// TwinCAT 3 PLC project Main
// ProgramVersion: 3.1.4022.4
// libraries:
//   Tc2_FTP, * (Beckhoff Automation GmbH)
//   Tc2_MC2, * (Beckhoff Automation GmbH)
//   Tc2_NCI, * (Beckhoff Automation GmbH)
//   Tc2_Standard, * (Beckhoff Automation GmbH)
//   Tc2_System, * (Beckhoff Automation GmbH)
//   Tc2_Utilities, * (Beckhoff Automation GmbH)
//   Tc3_IotBase, * (Beckhoff Automation GmbH)
//   Tc3_JsonXml, * (Beckhoff Automation GmbH)
//   Tc3_Module, * (Beckhoff Automation GmbH)
//   VisuSymbols,3.5.10.0,System
// project tree:
//   / GlobalTextList.TcGTLO, PlcTask.TcTTO, Visualization Manager.TcVMO (not stored)
//   GVLs/ COM.TcGVL, gcode.TcGVL, GVL.TcGVL
//   POUs/COMMANDS/ commandDecoder.TcPOU, commandExecute.TcPOU, POU_NCI.TcPOU
//   POUs/ ERROR.TcPOU, knoppen.TcPOU, MAIN_XYZ.TcPOU
//   POUs/JSON/ decCOM.TcPOU, decCOM_PLC.TcPOU, decFile.TcPOU, readJSONfile.TcPOU
//   POUs/MQTT/ MAIN_MQTT.TcPOU, PrgMqttCom.TcPOU, SubMqttCom.TcPOU
//   VISUs/ Basic.TcVIS, bStopAll.TcVIS, vKnoppen.TcVIS
// real-time tasks:
//   TASK PlcTask: cycle T#10ms, priority 20, ADS port 350
// motion (NC):
//   TASK NC-Task 1 SAF: cycle T#2ms, priority 4, ADS port 501
//   TASK NC-Task 1 SVB: cycle T#10ms, priority 8, ADS port 511
//   AXIS Axis X1 (id 1)
//     OtherSettings: AllowMotionCmdToSlave=true
//     encoder EncType=4
//       EncPara: ScaleFactorNumerator=40, ScaleFactorDenominator=12800, Inverse=true, MaxCount=#x0000ffff
//         SoftEndMinControl: Enable=true
//         SoftEndMaxControl: Enable=true, Range=275
//         Inc: RefSearchInverse=true, RefSyncInverse=false, RefMode=1, RefSoftSyncMask=#x0000ffff
//     drive DrvType=24
//       DrvPara: Inverse=true
//         Analog: VeloReferenz=400, ScaleFactorActTorque=0.1
//         TimeComp: TaskDelayCycles=1
//     controller CtrType=1
//       CtrPara: PriorControlFactor=1
//         PID: PosKp=25
//         Observer: BandWidth=20
//   AXIS Axis X2 (id 2)
//     OtherSettings: AllowMotionCmdToSlave=true
//     encoder EncType=4
//       EncPara: ScaleFactorNumerator=40, ScaleFactorDenominator=12800, Inverse=true, MaxCount=#x0000ffff
//         Inc: RefSoftSyncMask=#x0000ffff
//     drive DrvType=24
//       DrvPara: Inverse=true
//         Analog: VeloReferenz=400, ScaleFactorActTorque=0.1
//         TimeComp: TaskDelayCycles=1
//     controller CtrType=1
//       CtrPara: PriorControlFactor=1
//         PID: PosKp=25
//         Observer: BandWidth=20
//   AXIS Axis Y (id 4)
//     OtherSettings: AllowMotionCmdToSlave=true
//     encoder EncType=4
//       EncPara: ScaleFactorNumerator=40, ScaleFactorDenominator=12800, Inverse=true, MaxCount=#x0000ffff
//         SoftEndMinControl: Enable=true
//         SoftEndMaxControl: Enable=true, Range=275
//         Inc: RefSearchInverse=true, RefSyncInverse=false, RefMode=1, RefSoftSyncMask=#x0000ffff
//     drive DrvType=24
//       DrvPara: Inverse=true
//         Analog: VeloReferenz=400, ScaleFactorActTorque=0.1
//         TimeComp: TaskDelayCycles=1
//     controller CtrType=1
//       CtrPara: PriorControlFactor=1
//         PID: PosKp=25
//         Observer: BandWidth=20
//   AXIS Axis Z (id 3)
//     Velo: SlowManual=2, FastManual=5
//     OtherSettings: AllowMotionCmdToSlave=true
//     encoder EncType=4
//       EncPara: ScaleFactorNumerator=1, ScaleFactorDenominator=12800, MaxCount=#x0000ffff
//         Inc: RefSoftSyncMask=#x0000ffff
//     drive DrvType=24
//       Analog: VeloReferenz=10, ScaleFactorActTorque=0.1
//       TimeComp: TaskDelayCycles=1
//     controller CtrType=1
//       CtrPara: PriorControlFactor=1
//         PID: PosKp=25
//         Observer: BandWidth=20
// I/O:
//   DEVICE Device 3 (EtherCAT), AmsNetId 192.168.0.108.4.1
//     Term 1 (EK1100) [EK1100 EtherCAT Coupler (2A E-Bus)]
//       Term 2 (EL7031-0030) [EL7031-0030 1Ch. Stepper motor output stage (24V, 2.8A)]
//       Term 3 (EL7031-0030) [EL7031-0030 1Ch. Stepper motor output stage (24V, 2.8A)]
//       Term 4 (EL7031-0030) [EL7031-0030 1Ch. Stepper motor output stage (24V, 2.8A)]
//       Term 5 (EL7031-0030) [EL7031-0030 1Ch. Stepper motor output stage (24V, 2.8A)]
//       Term 6 (EL1008) [EL1008 8Ch. Dig. Input 24V, 3ms]
//       Term 14 (EL2008) [EL2008 8Ch. Dig. Output 24V, 0.5A]
//       Term 15 (EL3062) [EL3062 2Ch. Ana. Input 0-10V]
//       Term 7 (EL9011) [EL9011 End Terminal]
// variable links:
//   NC-Task 1 SAF/Axes/Axis X1 <-> Device 3 (EtherCAT)/Term 1 (EK1100)/Term 2 (EL7031-0030)
//     Drive/Inputs/In/nState1 @bit 3 <-> STM Status/Status/Error
//     Drive/Inputs/In/nState1 @bit 5 <-> STM Status/Status/Moving negative
//     Drive/Inputs/In/nState1 @bit 4 <-> STM Status/Status/Moving positive
//     Drive/Inputs/In/nState1 @bit 1 <-> STM Status/Status/Ready
//     Drive/Inputs/In/nState1 <-> STM Status/Status/Ready to enable
//     Drive/Inputs/In/nState1 @bit 6 <-> STM Status/Status/Torque reduced
//     Drive/Inputs/In/nState1 @bit 2 <-> STM Status/Status/Warning
//     Drive/Inputs/In/nState2 @bit 3 <-> STM Status/Status/Digital input 1
//     Drive/Inputs/In/nState2 @bit 4 <-> STM Status/Status/Digital input 2
//     Drive/Inputs/In/nState2 @bit 5 <-> STM Status/Status/Sync error
//     Drive/Inputs/In/nState2 @bit 7 <-> STM Status/Status/TxPDO Toggle
//     Drive/Inputs/In/nState4 @bit 1 <-> WcState/InputToggle
//     Drive/Inputs/In/nState4 <-> WcState/WcState
//     Drive/Outputs/Out/nCtrl1 <-> STM Control/Control/Enable
//     Drive/Outputs/Out/nCtrl1 @bit 2 <-> STM Control/Control/Reduce torque
//     Drive/Outputs/Out/nCtrl1 @bit 1 <-> STM Control/Control/Reset
//     Drive/Outputs/Out/nDataOut2[0] <-> STM Velocity/Velocity
//     Enc/Inputs/In/nDataIn1[0] <-> ENC Status compact/Counter value
//     Enc/Inputs/In/nDataIn2[0] <-> ENC Status compact/Latch value
//     Enc/Inputs/In/nState1 @bit 4 <-> ENC Status compact/Status/Counter overflow
//     Enc/Inputs/In/nState1 @bit 3 <-> ENC Status compact/Status/Counter underflow
//     Enc/Inputs/In/nState1 @bit 1 <-> ENC Status compact/Status/Latch extern valid
//     Enc/Inputs/In/nState1 @bit 2 <-> ENC Status compact/Status/Set counter done
//     Enc/Inputs/In/nState2 @bit 4 <-> ENC Status compact/Status/Status of extern latch
//     Enc/Inputs/In/nState2 @bit 5 <-> ENC Status compact/Status/Sync error
//     Enc/Inputs/In/nState2 @bit 7 <-> ENC Status compact/Status/TxPDO Toggle
//     Enc/Inputs/In/nState4 @bit 1 <-> WcState/InputToggle
//     Enc/Inputs/In/nState4 <-> WcState/WcState
//     Enc/Outputs/Out/nCtrl1 @bit 3 <-> ENC Control compact/Control/Enable latch extern on negative edge
//     Enc/Outputs/Out/nCtrl1 @bit 1 <-> ENC Control compact/Control/Enable latch extern on positive edge
//     Enc/Outputs/Out/nCtrl1 @bit 2 <-> ENC Control compact/Control/Set counter
//     Enc/Outputs/Out/nDataOut1[0] <-> ENC Control compact/Set counter value
//   NC-Task 1 SAF/Axes/Axis X2 <-> Device 3 (EtherCAT)/Term 1 (EK1100)/Term 3 (EL7031-0030)
//     Drive/Inputs/In/nState1 @bit 3 <-> STM Status/Status/Error
//     Drive/Inputs/In/nState1 @bit 5 <-> STM Status/Status/Moving negative
//     Drive/Inputs/In/nState1 @bit 4 <-> STM Status/Status/Moving positive
//     Drive/Inputs/In/nState1 @bit 1 <-> STM Status/Status/Ready
//     Drive/Inputs/In/nState1 <-> STM Status/Status/Ready to enable
//     Drive/Inputs/In/nState1 @bit 6 <-> STM Status/Status/Torque reduced
//     Drive/Inputs/In/nState1 @bit 2 <-> STM Status/Status/Warning
//     Drive/Inputs/In/nState2 @bit 3 <-> STM Status/Status/Digital input 1
//     Drive/Inputs/In/nState2 @bit 4 <-> STM Status/Status/Digital input 2
//     Drive/Inputs/In/nState2 @bit 5 <-> STM Status/Status/Sync error
//     Drive/Inputs/In/nState2 @bit 7 <-> STM Status/Status/TxPDO Toggle
//     Drive/Inputs/In/nState4 @bit 1 <-> WcState/InputToggle
//     Drive/Inputs/In/nState4 <-> WcState/WcState
//     Drive/Outputs/Out/nCtrl1 <-> STM Control/Control/Enable
//     Drive/Outputs/Out/nCtrl1 @bit 2 <-> STM Control/Control/Reduce torque
//     Drive/Outputs/Out/nCtrl1 @bit 1 <-> STM Control/Control/Reset
//     Drive/Outputs/Out/nDataOut2[0] <-> STM Velocity/Velocity
//     Enc/Inputs/In/nDataIn1[0] <-> ENC Status compact/Counter value
//     Enc/Inputs/In/nDataIn2[0] <-> ENC Status compact/Latch value
//     Enc/Inputs/In/nState1 @bit 4 <-> ENC Status compact/Status/Counter overflow
//     Enc/Inputs/In/nState1 @bit 3 <-> ENC Status compact/Status/Counter underflow
//     Enc/Inputs/In/nState1 @bit 1 <-> ENC Status compact/Status/Latch extern valid
//     Enc/Inputs/In/nState1 @bit 2 <-> ENC Status compact/Status/Set counter done
//     Enc/Inputs/In/nState2 @bit 4 <-> ENC Status compact/Status/Status of extern latch
//     Enc/Inputs/In/nState2 @bit 5 <-> ENC Status compact/Status/Sync error
//     Enc/Inputs/In/nState2 @bit 7 <-> ENC Status compact/Status/TxPDO Toggle
//     Enc/Inputs/In/nState4 @bit 1 <-> WcState/InputToggle
//     Enc/Inputs/In/nState4 <-> WcState/WcState
//     Enc/Outputs/Out/nCtrl1 @bit 3 <-> ENC Control compact/Control/Enable latch extern on negative edge
//     Enc/Outputs/Out/nCtrl1 @bit 1 <-> ENC Control compact/Control/Enable latch extern on positive edge
//     Enc/Outputs/Out/nCtrl1 @bit 2 <-> ENC Control compact/Control/Set counter
//     Enc/Outputs/Out/nDataOut1[0] <-> ENC Control compact/Set counter value
//   NC-Task 1 SAF/Axes/Axis Y <-> Device 3 (EtherCAT)/Term 1 (EK1100)/Term 5 (EL7031-0030)
//     Drive/Inputs/In/nState1 @bit 3 <-> STM Status/Status/Error
//     Drive/Inputs/In/nState1 @bit 5 <-> STM Status/Status/Moving negative
//     Drive/Inputs/In/nState1 @bit 4 <-> STM Status/Status/Moving positive
//     Drive/Inputs/In/nState1 @bit 1 <-> STM Status/Status/Ready
//     Drive/Inputs/In/nState1 <-> STM Status/Status/Ready to enable
//     Drive/Inputs/In/nState1 @bit 6 <-> STM Status/Status/Torque reduced
//     Drive/Inputs/In/nState1 @bit 2 <-> STM Status/Status/Warning
//     Drive/Inputs/In/nState2 @bit 3 <-> STM Status/Status/Digital input 1
//     Drive/Inputs/In/nState2 @bit 4 <-> STM Status/Status/Digital input 2
//     Drive/Inputs/In/nState2 @bit 5 <-> STM Status/Status/Sync error
//     Drive/Inputs/In/nState2 @bit 7 <-> STM Status/Status/TxPDO Toggle
//     Drive/Inputs/In/nState4 @bit 1 <-> WcState/InputToggle
//     Drive/Inputs/In/nState4 <-> WcState/WcState
//     Drive/Outputs/Out/nCtrl1 <-> STM Control/Control/Enable
//     Drive/Outputs/Out/nCtrl1 @bit 2 <-> STM Control/Control/Reduce torque
//     Drive/Outputs/Out/nCtrl1 @bit 1 <-> STM Control/Control/Reset
//     Drive/Outputs/Out/nDataOut2[0] <-> STM Velocity/Velocity
//     Enc/Inputs/In/nDataIn1[0] <-> ENC Status compact/Counter value
//     Enc/Inputs/In/nDataIn2[0] <-> ENC Status compact/Latch value
//     Enc/Inputs/In/nState1 @bit 4 <-> ENC Status compact/Status/Counter overflow
//     Enc/Inputs/In/nState1 @bit 3 <-> ENC Status compact/Status/Counter underflow
//     Enc/Inputs/In/nState1 @bit 1 <-> ENC Status compact/Status/Latch extern valid
//     Enc/Inputs/In/nState1 @bit 2 <-> ENC Status compact/Status/Set counter done
//     Enc/Inputs/In/nState2 @bit 4 <-> ENC Status compact/Status/Status of extern latch
//     Enc/Inputs/In/nState2 @bit 5 <-> ENC Status compact/Status/Sync error
//     Enc/Inputs/In/nState2 @bit 7 <-> ENC Status compact/Status/TxPDO Toggle
//     Enc/Inputs/In/nState4 @bit 1 <-> WcState/InputToggle
//     Enc/Inputs/In/nState4 <-> WcState/WcState
//     Enc/Outputs/Out/nCtrl1 @bit 3 <-> ENC Control compact/Control/Enable latch extern on negative edge
//     Enc/Outputs/Out/nCtrl1 @bit 1 <-> ENC Control compact/Control/Enable latch extern on positive edge
//     Enc/Outputs/Out/nCtrl1 @bit 2 <-> ENC Control compact/Control/Set counter
//     Enc/Outputs/Out/nDataOut1[0] <-> ENC Control compact/Set counter value
//   NC-Task 1 SAF/Axes/Axis Z <-> Device 3 (EtherCAT)/Term 1 (EK1100)/Term 4 (EL7031-0030)
//     Drive/Inputs/In/nState1 @bit 3 <-> STM Status/Status/Error
//     Drive/Inputs/In/nState1 @bit 5 <-> STM Status/Status/Moving negative
//     Drive/Inputs/In/nState1 @bit 4 <-> STM Status/Status/Moving positive
//     Drive/Inputs/In/nState1 @bit 1 <-> STM Status/Status/Ready
//     Drive/Inputs/In/nState1 <-> STM Status/Status/Ready to enable
//     Drive/Inputs/In/nState1 @bit 6 <-> STM Status/Status/Torque reduced
//     Drive/Inputs/In/nState1 @bit 2 <-> STM Status/Status/Warning
//     Drive/Inputs/In/nState2 @bit 3 <-> STM Status/Status/Digital input 1
//     Drive/Inputs/In/nState2 @bit 4 <-> STM Status/Status/Digital input 2
//     Drive/Inputs/In/nState2 @bit 5 <-> STM Status/Status/Sync error
//     Drive/Inputs/In/nState2 @bit 7 <-> STM Status/Status/TxPDO Toggle
//     Drive/Inputs/In/nState4 @bit 1 <-> WcState/InputToggle
//     Drive/Inputs/In/nState4 <-> WcState/WcState
//     Drive/Outputs/Out/nCtrl1 <-> STM Control/Control/Enable
//     Drive/Outputs/Out/nCtrl1 @bit 2 <-> STM Control/Control/Reduce torque
//     Drive/Outputs/Out/nCtrl1 @bit 1 <-> STM Control/Control/Reset
//     Drive/Outputs/Out/nDataOut2[0] <-> STM Velocity/Velocity
//     Enc/Inputs/In/nDataIn1[0] <-> ENC Status compact/Counter value
//     Enc/Inputs/In/nDataIn2[0] <-> ENC Status compact/Latch value
//     Enc/Inputs/In/nState1 @bit 4 <-> ENC Status compact/Status/Counter overflow
//     Enc/Inputs/In/nState1 @bit 3 <-> ENC Status compact/Status/Counter underflow
//     Enc/Inputs/In/nState1 @bit 1 <-> ENC Status compact/Status/Latch extern valid
//     Enc/Inputs/In/nState1 @bit 2 <-> ENC Status compact/Status/Set counter done
//     Enc/Inputs/In/nState2 @bit 4 <-> ENC Status compact/Status/Status of extern latch
//     Enc/Inputs/In/nState2 @bit 5 <-> ENC Status compact/Status/Sync error
//     Enc/Inputs/In/nState2 @bit 7 <-> ENC Status compact/Status/TxPDO Toggle
//     Enc/Inputs/In/nState4 @bit 1 <-> WcState/InputToggle
//     Enc/Inputs/In/nState4 <-> WcState/WcState
//     Enc/Outputs/Out/nCtrl1 @bit 3 <-> ENC Control compact/Control/Enable latch extern on negative edge
//     Enc/Outputs/Out/nCtrl1 @bit 1 <-> ENC Control compact/Control/Enable latch extern on positive edge
//     Enc/Outputs/Out/nCtrl1 @bit 2 <-> ENC Control compact/Control/Set counter
//     Enc/Outputs/Out/nDataOut1[0] <-> ENC Control compact/Set counter value
//   Main/Main Instance <-> Device 3 (EtherCAT)/Term 1 (EK1100)/Term 6 (EL1008)
//     PlcTask Inputs/GVL.bX1 <-> Channel 3/Input
//     PlcTask Inputs/GVL.bX2 <-> Channel 4/Input
//     PlcTask Inputs/GVL.bY1 <-> Channel 1/Input
//     PlcTask Inputs/GVL.bY2 <-> Channel 2/Input
//   Main/Main Instance <-> NC-Task 1 SAF/Axes/Axis X1
//     PlcTask Inputs/GVL.As_Xa.NcToPlc <-> Outputs/ToPlc
//     PlcTask Outputs/GVL.As_Xa.PlcToNc <-> Inputs/FromPlc
//   Main/Main Instance <-> NC-Task 1 SAF/Axes/Axis X2
//     PlcTask Inputs/GVL.As_Xb.NcToPlc <-> Outputs/ToPlc
//     PlcTask Outputs/GVL.As_Xb.PlcToNc <-> Inputs/FromPlc
//   Main/Main Instance <-> NC-Task 1 SAF/Axes/Axis Y
//     PlcTask Inputs/GVL.As_Y.NcToPlc <-> Outputs/ToPlc
//     PlcTask Outputs/GVL.As_Y.PlcToNc <-> Inputs/FromPlc
//   Main/Main Instance <-> NC-Task 1 SAF/Axes/Axis Z
//     PlcTask Inputs/GVL.As_Z.NcToPlc <-> Outputs/ToPlc
//     PlcTask Outputs/GVL.As_Z.PlcToNc <-> Inputs/FromPlc
//   Main/Main Instance <-> NC-Task 1 SAF/G-code
//     PlcTask Inputs/GVL.ChannelInput <-> Outputs/ToPlc
//     PlcTask Outputs/GVL.ChannelOutput <-> Inputs/FromPlc

CONFIGURATION Main
    RESOURCE PLC ON TwinCAT3
        TASK PlcTask(INTERVAL := T#10ms, PRIORITY := 20);
        PROGRAM MAIN_XYZ WITH PlcTask : MAIN_XYZ;
    END_RESOURCE
END_CONFIGURATION

// ---- GVLs/COM.TcGVL
{attribute 'qualified_only'}
VAR_GLOBAL
	bEnable			: BOOL := FALSE;
	bCouple			: BOOL := FALSE;
	bReset			: BOOL := FALSE;
	bHome			: BOOL := FALSE;
	
	bMoveX			: BOOL;
	bMoveY			: BOOL;
	bMoveZ			: BOOL;
	bRelZ			: BOOL;
	bSetZ			: BOOL;
	
	bValid			: BOOL;
	bHomeDone		: BOOL;
	bHomeBusy		: BOOL;
	bMoveDone		: BOOL;
	bMoveXDone		: BOOL;
	bMoveYDone		: BOOL;
	bMoveZDone		: BOOL;
	bMoveZRelDone   : BOOL;
	bMoveBusy		: BOOL;
	bError 			: BOOL;	
	
	inUSe 			: BOOL;
	IFerror			: BOOL;
	
	JSONFromFile 	: STRING(2047);
	JSONFILE		: STRING (2047);
	sendCommand 	: STRING;
	
	Xval			: INT;
	Yval			: INT;
	Zval			: INT;
	
	goX				: INT := 10;
	goY				: INT := 10;
	goZ				: INT := 10;
	
	object1			: INT := 0;
	object2			: INT := 0;
	
	absX 			: INT := 0;
	absY 			: INT := 0;
	absZ 			: INT := 0;
	relZ   			: INT := 0;
	            	
	velX 			: INT := 100;	//0-400
	velY 			: INT := 100;	//0-400
	velZ 			: INT := 2;		//0-10
	
	PosX 			: LREAL;
	PosY 			: LREAL;
	PosZ 			: LREAL;
	
	objectNum		: INT := 1;
	objectread		: BOOL;
	objectx			: LREAL;
	objecty			: LREAL;
	readfile        : BOOL;
	
END_VAR

// ---- GVLs/gcode.TcGVL
{attribute 'qualified_only'}
VAR_GLOBAL
	bBuildGroup	: BOOL;
	bLoad		: BOOL;
	bStart		: BOOL;
	bStop		: BOOL;
	bReset		: BOOL;
END_VAR

// ---- GVLs/GVL.TcGVL
{attribute 'qualified_only'}
VAR_GLOBAL
	As_Xa : AXIS_REF;
	As_Xb : AXIS_REF;
	As_Y : AXIS_REF;
	As_Z : AXIS_REF;
	
	ChannelInput AT %I* : NCTOPLC_NCICHANNEL_REF;
	ChannelOutput AT %Q* : PLCTONC_NCICHANNEL_REF;
	
	StopALL : bool;
	
	bX1 AT%I* : BOOL;
	bX2 AT%I* : BOOL;
	bY1 AT%I* : BOOL;
	bY2 AT%I* : BOOL;
	
	stReceivedData	: STRING(255);
		//-------------------------
	message_sub : STRING(2047);
	message_pub : STRING(2047);
	message_PayLoad : STRING(2047);
	
	// FLAGS
	flag_pub : BOOL := FALSE;
	flag_sub : BOOL := FALSE;
	
	bSendMessage : BOOL;
	
	configHoming	: BOOL := FALSE;
	configZaxis		: BOOL := FALSE;
END_VAR

// ---- POUs/MAIN_XYZ.TcPOU
PROGRAM MAIN_XYZ
VAR
	
END_VAR

//main program for gcode
	//POU_NCI();

//JSON
	decCOM();
	readJSONfile();
	decFile();

//AT Commands
	commandDecoder();
	commandExecute();

//Error
	ERROR();

MAIN_MQTT();

END_PROGRAM

// ---- POUs/JSON/decCOM.TcPOU
PROGRAM decCOM
VAR
	recString 			: STRING(2047);
	RisingEdge         : R_TRIG;
	bExecute			: BOOL;
	bReset				: BOOL;

	fbJson 				: FB_JsonDomParser;
                    	
	jsonDoc 			: SJsonValue;
	jsonDoc2 			: SJsonValue;
	                	
	jsonProp			: SJsonValue;
	jsonProp2			: SJsonValue;           	

	jsontempval			: SJsonValue;
	
	getInput			: STRING(2047);
	getRawValue 		: STRING;
	getValueStr 		: STRING;
	getValue1			: STRING(2047);
	
	jsonGetulint		: ULINT;
	jsongettype			: Tc3_JsonXml.EJsonType;
	jsongetArraySize	: UDINT;
	jsongetArray		: ARRAY[0..1000] OF SJsonValue;
	jsongetArrayulint	: ULINT;
	jsongetArrayudint	: UDINT;
	
	JSONTEMP			: STRING(2047);
	
	JSONVal1 			: STRING;
	JSONVal2 			: STRING;
	JSONVal3 			: STRING;
	JSONVal4 			: STRING;
	JSONVal5 			: STRING;
	JSONVal6 			: STRING;
	
	cnt : UDINT;	
	temp : string;
END_VAR

RisingEdge(CLK:=bReset);
IF RisingEdge.Q THEN
	JSONVal1	:= '';
	JSONVal2	:= '';
	JSONVal3	:= '';
    JSONVal4	:= '';
    JSONVal5	:= '';
    JSONVal6	:= '';
	bReset 		:= FALSE;
END_IF

IF NOT(GVL.message_sub = '') THEN
	recString := GVL.message_sub;
	jsonDoc := fbJson.ParseDocument(recString);
	
	jsonProp := fbJson.FindMember(jsonDoc, 'slots');
	cnt := 0;
	 
	IF (jsonProp <> 0) THEN
		jsongettype			:= fbJson.GetType(jsonProp);
		jsongetArraySize	:= fbJson.GetArraySize(jsonProp);
		FOR cnt := 0 TO jsongetArraySize-1 BY 1 DO
			jsontempval		:= fbJson.GetArrayValueByIdx(jsonProp, cnt);
			JSONTEMP				:= fbJson.GetJson( jsontempval );
				jsonDoc2 			:= fbJson.ParseDocument(JSONTEMP);
				jsonProp2 			:= fbJson.FindMember(jsonDoc2, 'value');
					jsonProp2 		:= fbJson.FindMember(jsonProp2, 'value');
						CASE cnt OF
							0:	JSONVal1	:= fbJson.GetString(jsonProp2);
							1:	JSONVal2	:= fbJson.GetString(jsonProp2);
							2:	JSONVal3	:= fbJson.GetString(jsonProp2);
							3:	JSONVal4	:= fbJson.GetString(jsonProp2);
							4:	JSONVal5	:= fbJson.GetString(jsonProp2);
							5:	JSONVal6	:= fbJson.GetString(jsonProp2);
						END_CASE
		END_FOR
		
		CASE cnt OF
			1:
				IF 		(JSONVal1 = 'Do homing') 						THEN							com.sendCommand := 'do homing';				
				ELSIF 	(JSONVal1 = 'Execute trace') 					THEN							com.sendCommand := 'execute trace';			
				ELSIF 	(JSONVal1 = 'Execute sort') 					THEN							com.sendCommand := 'execute sort';
				ELSIF 	(JSONVal1 = 'Execute Drill') 					THEN							com.sendCommand := 'execute drill';
				ELSIF 	(JSONVal1 = 'Stop') 							THEN							com.sendCommand := 'stop';	
				ELSIF 	(JSONVal1 = 'z to zero') 						THEN							com.sendCommand := 'z to zero';
				ELSIF 	(JSONVal1 = 'read position') 					THEN							com.sendCommand := 'read position';	
				ELSIF 	(JSONVal1 = 'read error') 						THEN							com.sendCommand := 'read error';	
				ELSIF 	(JSONVal1 = 'read files') 						THEN							com.sendCommand := 'read files';	
				ELSIF 	(JSONVal1 = 'execute Gcode')					THEN							com.sendCommand := 'execute gcode';	
				ELSIF 	(JSONVal1 = 'reset') 							THEN							com.sendCommand := 'reset';	
				END_IF
			2:
				IF 		(JSONVal1 = 'show difference') 					THEN							com.sendCommand := 'show difference';
																										com.object1		:= STRING_TO_INT(JSONVal2);	
				ELSIF 	(JSONVal1 = 'show object') 						THEN							com.sendCommand := 'show object';
																										com.object1		:= STRING_TO_INT(JSONVal2);	
				ELSIF 	(JSONVal1 = 'delete difference') 				THEN							com.sendCommand := 'delete difference';
																										com.object1		:= STRING_TO_INT(JSONVal2);	
				ELSIF 	(JSONVal1 = 'turn difference') 					THEN							com.sendCommand := 'turn difference';
																										com.object1		:= STRING_TO_INT(JSONVal2);
				ELSIF 	(JSONVal1 = 'turn object') 						THEN							com.sendCommand := 'turn object';
																										com.object1		:= STRING_TO_INT(JSONVal2);
				ELSIF 	(JSONVal1 = 'X-axis') 							THEN							com.sendCommand := 'x-axis';
																										com.goX		:= STRING_TO_INT(JSONVal2);
				ELSIF 	(JSONVal1 = 'Y-axis') 							THEN							com.sendCommand := 'y-axis';
																										com.goY		:= STRING_TO_INT(JSONVal2);
				ELSIF 	(JSONVal1 = 'Z-axis') 							THEN							com.sendCommand := 'z-axis';
																										com.goZ		:= STRING_TO_INT(JSONVal2);
				ELSIF 	(JSONVal1 = 'Up') 								THEN							com.sendCommand := 'Up';
																										com.goZ		:= STRING_TO_INT(JSONVal2);
				ELSIF 	(JSONVal1 = 'Down') 							THEN							com.sendCommand := 'Down';
																										com.goZ		:= STRING_TO_INT(JSONVal2);					
				END_IF
			4:
				IF 		(JSONVal1 = 'X-axis' AND JSONVal3 = 'Y-axis')	THEN 							com.sendCommand := 'go xy';
																										com.goX			:= STRING_TO_INT(JSONVal2);	
																										com.goY			:= STRING_TO_INT(JSONVal4);		
				ELSIF 	(JSONVal1 = 'combine difference') 				THEN							com.sendCommand := 'combine difference';
																										com.object1		:= STRING_TO_INT(JSONVal2);	
																										com.object2		:= STRING_TO_INT(JSONVal4);
				ELSIF 	(JSONVal1 = 'combine object') 					THEN							com.sendCommand := 'combine object';
																										com.object1		:= STRING_TO_INT(JSONVal2);	
																										com.object2		:= STRING_TO_INT(JSONVal4);
				END_IF													
			6:
				IF 		(JSONVal1 = 'X-axis' AND JSONVal3 = 'Y-axis' AND JSONVal5 = 'Z-axis') THEN		com.sendCommand := 'go xyz';
																										com.goX			:= STRING_TO_INT(JSONVal2);	
																										com.goY			:= STRING_TO_INT(JSONVal4);
																										com.goZ			:= STRING_TO_INT(JSONVal6);
				END_IF
		END_CASE
	END_IF
	GVL.message_sub := '';
	temp := recString;
	recString := '';
END_IF

END_PROGRAM

// ---- POUs/ERROR.TcPOU
PROGRAM ERROR
VAR
	StopX_a : MC_Stop;
	StopX_b : MC_Stop;
	StopY 	: MC_Stop;
	StopZ 	: MC_Stop;
	
	FB_AXISERRORXa, FB_AXISERRORXb, FB_AXISERRORY, FB_AXISERRORZ : MC_ReadAxisError;
	
	ErrorIDXa 	: DWORD;
	ErrorIDXb 	: DWORD;
	ErrorIDY 	: DWORD;
	ErrorIDZ 	: DWORD;
	
	ErrorAxisXa	: UDINT;
	ErrorAxisXb	: UDINT;
	ErrorAxisY	: UDINT;
	ErrorAxisZ	: UDINT;
END_VAR

//stop all
StopX_a(Axis := gvl.As_Xa,
		Execute := GVL.StopALL);

StopX_b(Axis := gvl.As_Xb,
		Execute := GVL.StopALL);

StopY(Axis := gvl.As_Y,
		Execute := GVL.StopALL);
		
StopZ(Axis := gvl.As_Z,
		Execute := GVL.StopALL);

//error		
FB_AxisErrorXa(Axis := gvl.As_Xa, Enable := TRUE);
FB_AxisErrorXb(Axis := gvl.As_Xb, Enable := TRUE);
FB_AxisErrorY (Axis := gvl.As_Y,  Enable := TRUE);
FB_AxisErrorZ (Axis := gvl.As_Z,  Enable := TRUE);

ErrorIDXa 	:= FB_AxisErrorXa.ErrorID;
ErrorIDXb 	:= FB_AxisErrorXb.ErrorID;
ErrorIDY 	:= FB_AxisErrorY.ErrorID;
ErrorIDZ 	:= FB_AxisErrorZ.ErrorID;

ErrorAxisXa	:= FB_AxisErrorXa.AxisErrorID;
ErrorAxisXb	:= FB_AxisErrorXb.AxisErrorID;
ErrorAxisY	:= FB_AxisErrorY.AxisErrorID;
ErrorAxisZ	:= FB_AxisErrorZ.AxisErrorID;

com.IFerror := FB_axiserrorxa.Error OR FB_axiserrorxb.Error OR FB_axiserrory.Error OR FB_axiserrorz.Error;

END_PROGRAM

// ---- POUs/JSON/readJSONfile.TcPOU
PROGRAM readJSONfile
VAR
		sSrcNetId		        : T_AmsNetId := '';						(* TwinCAT network address of the source file *)
		
		sSrcPathName            : T_MaxString:=  'C:\Users\Jarni\OneDrive - PXL\Engineering Project\cedric\test.json';	
	
        bExecute                : BOOL; 								(* Rising edge start fb execution *)
        tTimeOut                : TIME := DEFAULT_ADS_TIMEOUT;			(* Max. ADS timeout time *)

        bBusy                   : BOOL;									(* TRUE => File copy execution in progress, FALSE => File copy execution idle *)
	 	bError                  : BOOL;									(* TRUE => Error, FALSE => No error *)
	 	nErrId                  : UDINT;								(* Error code *)

        fbFileOpen              : FB_FileOpen;
        fbFileClose             : FB_FileClose;
        fbFileRead              : FB_FileRead;
        fbFileWrite             : FB_FileWrite;

        hSrcFile                : UINT   := 0;							(* File handle of the source file *)
 		hDestFile               : UINT   := 0;							(* File handle of the destination file *)

        Step                    : DWORD;									(* For Case*)
        RisingEdge              : R_TRIG;

        buffRead                : STRING(2047);    						(* String read from file, JSON CODE *)
		findN					: STRING := '$N';  						(* String to replace *)
		findT					: STRING := '$T';  						(* String to replace *)
		replstr					: STRING := '';    						(* Replace with '' *)
 		cbReadLength            : UDINT := 0;	    					(* *)				

END_VAR

RisingEdge(CLK:=bExecute OR com.readfile );

CASE Step OF
        0:      (* Idle state *)
         	IF RisingEdge.Q THEN
                        bBusy := TRUE;
                        bError:= FALSE;
                        nErrId:=0;
                        Step := 1;
                        cbReadLength:=0;
                        hSrcFile:=0;
                        hDestFile:=0;
                END_IF

        1:      (* Open source file *)
			fbFileOpen( bExecute := FALSE );
			fbFileOpen( sNetId := sSrcNetId, sPathName := sSrcPathName,				//temporary static
					nMode := FOPEN_MODEREAD OR FOPEN_MODETEXT,
					ePath := PATH_GENERIC, tTimeout := tTimeOut, bExecute := TRUE );
			Step := Step + 1;
				
        2:		(* Check for erros *)    
			fbFileOpen( bExecute := FALSE );
			IF NOT fbFileOpen.bBusy THEN
					IF fbFileOpen.bError THEN
							nErrId := fbFileOpen.nErrId;
							bError := TRUE;
							Step := 50;
					ELSE
							hSrcFile := fbFileOpen.hFile;
							Step := Step + 1;
					END_IF
			END_IF

		3:      (* Read data from source file *)
			cbReadLength := 0;
			fbFileRead( bExecute:= FALSE );
			fbFileRead( bExecute:=TRUE, sNetId:=sSrcNetId, hFile:=hSrcFile,
					pReadBuff:= ADR(buffRead), cbReadLen:= SIZEOF(buffRead),
					tTimeout:=tTimeOut );
			Step := Step + 1;
				
		4:  	(* Check for erros *)    
			fbFileRead( bExecute:= FALSE );
			IF NOT fbFileRead.bBusy THEN
					IF fbFileRead.bError THEN
							nErrId := fbFileRead.nErrId;
							bError := TRUE;
							Step := 50;
					ELSE
							cbReadLength := fbFileRead.cbRead;
							Step := Step + 1;
					END_IF
			END_IF
				
		5:		(* Deletes "$N" AND "$T" in the string *)
			FindAndReplace( ADR(buffRead), ADR(findN), ADR(replstr), ADR(buffRead), SIZEOF(buffRead) );  //$N
			FindAndReplace( ADR(buffRead), ADR(findT), ADR(replstr), ADR(buffRead), SIZEOF(buffRead) );	 //$T
			COM.JSONFILE := buffRead;  
			Step := 50;
		
        40:		(* Close source file *)
			fbFileClose( bExecute := FALSE );
			fbFileClose( sNetId:=sSrcNetId, hFile:=hSrcFile, bExecute:=TRUE, tTimeout:=tTimeOut );
			Step := Step + 1;
			
        41:		(* Check for erros *)    
			fbFileClose( bExecute := FALSE );
			IF NOT fbFileClose.bBusy THEN
					IF fbFileClose.bError THEN
							nErrId := fbFileClose.nErrId;
							bError := TRUE;
					END_IF
					Step := 50;
					hSrcFile := 0;
			END_IF

        50: (* Error or ready => Cleanup *)
			 IF (hSrcFile <> 0 ) THEN
							Step := 40; (* Close the source file *)
			 ELSE
							Step := 0;      (* Ready *)
							bBusy := FALSE;
			 END_IF
			 bexecute := FALSE;
			 com.readfile := FALSE;
END_CASE

END_PROGRAM

// ---- POUs/JSON/decFile.TcPOU
PROGRAM decFile
VAR
	s1 : STRING(2000);
	recString: STRING(2047);
	
	fbJson 				: FB_JsonDomParser;
	jsonDoc 			: SJsonValue;
	jsonDoc2 			: SJsonValue;
	jsonProp			: SJsonValue;
	jsonProp2			: SJsonValue;
	jsontempval			: SJsonValue;
	jsontempval2			: SJsonValue;
	jsongettype			: Tc3_JsonXml.EJsonType;
	jsonGetulint		: ULINT;
	jsongetArraySize	: UDINT;
	jsongetArray		: ARRAY[0..1000] OF SJsonValue;
	jsongetArrayulint	: ULINT;
	jsongetArrayudint	: UDINT;
	
	temp 				: STRING;
	btest				: BOOL;
	RisingEdge         : R_TRIG;
	
	JSONVal1 			: STRING;
	JSONVal2 			: STRING;
	
	JSONstr 			: STRING;
	getobj				: INT := 1;
	tempint				: INT;
	
	JSONTEMP			: STRING(2047);
END_VAR

s1 := com.JSONFile;
RisingEdge(CLK:=btest);

IF NOT(s1 = '' AND com.objectread) THEN
	jsonDoc := fbJson.ParseDocument(s1);
	jsonProp :=  fbJson.FindMember(jsonDoc, 'objects');;
	tempint := com.objectNum -1;
	
	IF (jsonProp <> 0) THEN
		jsongettype			:= fbJson.GetType(jsonProp);
		jsongetArraySize	:= fbJson.GetArraySize(jsonProp);
			jsontempval		:= fbJson.GetArrayValueByIdx(jsonProp, (INT_TO_UDINT (tempint) ) );
			JSONTEMP		:= fbJson.GetJson( jsontempval );
				jsonDoc2 			:= fbJson.ParseDocument(JSONTEMP);
				jsonProp2			:= fbJson.FindMember(jsonDoc2, 'centrepointy');
				JSONVal1 			:= fbJson.GetJson(jsonProp2);
				com.objectx			:= STRING_TO_LREAL(JSONVal1);
				
				jsonProp2			:= fbJson.FindMember(jsonDoc2, 'centrepointx');
				JSONVal2 			:= fbJson.GetJson(jsonProp2);
				com.objecty			:= STRING_TO_LREAL(JSONVal2);
	
	END_IF
	
	btest := false;
END_IF

END_PROGRAM

// ---- POUs/COMMANDS/commandDecoder.TcPOU
PROGRAM commandDecoder
VAR
	command 	: STRING(255);
	Head_Loaded : STRING;
	index 		: INT := 0;
	
	actualX 	: LREAL;
	actualY 	: LREAL;
	actualZ 	: Lreal;
	
	wait100ms : TON;
	wait200ms : TON;
	
END_VAR

wait100ms(IN := COM.bEnable OR gvl.StopALL, pt := T#500MS);
wait200ms(IN := COM.bEnable OR gvl.StopALL, pt := T#1S);

IF ( NOT (com.sendCommand = '') ) THEN
	command := F_ToLCase(com.sendCommand);
	com.sendCommand := '';
END_IF

CASE index OF
	0:	//commands
		COM.bEnable := FALSE;
		COM.bCouple := FALSE;
		COM.bHome 	:= FALSE;
		COM.inUSe 	:= FALSE;
		
		IF ( NOT (command = '') ) THEN
			IF 		(command = 'error' OR com.IFerror) THEN		index := 999;
			ELSIF 	(command = 'reset') THEN					index := 10;
			ELSIF 	(command = 'stop') THEN						index := 20;
			ELSIF 	(command = 'do homing') THEN				index := 100;
			ELSIF 	(command = 'z to zero') THEN				index := 110;
			ELSIF 	(command = 'go xyz') THEN					index := 200;
			ELSIF 	(command = 'go xy') THEN					index := 205;
			ELSIF 	(command = 'x-axis') THEN					index := 210;
			ELSIF 	(command = 'y-axis') THEN					index := 220;
			ELSIF 	(command = 'z-axis') THEN					index := 230;
			ELSIF 	(command = 'exec gcode') THEN				index := 250;
			ELSIF 	(command = 'execute trace') THEN			index := 260;
			ELSIF 	(command = 'execute sort') THEN				index := 270;
			ELSIF 	(command = 'execute drill') THEN			index := 280;
			ELSIF 	(command = 'read position') THEN			index := 300;
			ELSIF 	(command = 'up') THEN						index := 450;
			ELSIF 	(command = 'down') THEN						index := 460;
			ELSIF 	(command = 'show object') THEN				index := 600;
			ELSE												index := 0;
			END_IF;
			command := '';
		ELSE 
			index := 0;
		END_IF;
		
	10:  //reset
		GVL.message_pub  := '{"text": "Resetting"}';
		GVL.bSendMessage := TRUE;
	
		gcode.bReset := TRUE;
		COM.bReset 	:= TRUE;
		COM.bEnable := FALSE;
		COM.bCouple := FALSE;
		COM.bHome 	:= FALSE;
		COM.inUSe 	:= FALSE;
		COM.bMoveX 	:= FALSE;
		COM.bMoveY 	:= FALSE;
		COM.bMoveZ 	:= FALSE;
		COM.bReset 	:= FALSE;	
		gcode.bReset := FALSE;
		
		index 		:= 0;
		
	20:  //Stop
		gvl.StopALL := TRUE;
		
		GVL.message_pub  := '{"text": "Stopping program"}';
		GVL.bSendMessage := TRUE;
		
		IF wait100ms.q THEN
			gvl.StopALL := FALSE;
			index 		:= 0;
		END_IF
			
	100: //Do homing
		COM.bEnable := TRUE;
		COM.bCouple := TRUE;
		COM.bHome 	:= TRUE;
		
		GVL.message_pub  := '{"text": "Doing homing"}';
		GVL.bSendMessage := TRUE;
		
		IF COM.bHomeBusy THEN
			COM.inUSe 	:= TRUE;
		ELSE
			COM.inUSe 	:= FALSE;
		END_IF
		IF COM.bHomeDone THEN
			COM.bEnable := FALSE;
			COM.bCouple := FALSE;
			COM.bHome 	:= FALSE;
			COM.inUSe 	:= FALSE;
			gvl.configHoming := TRUE;
			index 	:= 0;
		END_IF
		
	110: //set Z position to zero
		COM.bSetZ 		:= TRUE;
		
		GVL.message_pub  := '{"text": "Z axis has been set to zero"}';
		GVL.bSendMessage := TRUE;
		
		IF (COM.PosZ = 0 AND COM.bValid) THEN
			COM.bSetZ 	:= FALSE;
			gvl.configZaxis := TRUE;
			index 		:= 0;
		END_IF
				
	200: //Go to xyz Pos
    	COM.absX := (COM.goX);
		COM.absY := (COM.goY);
		COM.absZ := (COM.goZ);
		
		IF gvl.configHoming THEN
			COM.bEnable := TRUE;
			COM.bCouple := TRUE;
			
			IF wait100ms.Q THEN 
				COM.bMoveX 	:= TRUE;
				COM.bMoveY 	:= TRUE;
				COM.bMoveZ 	:= TRUE;
			END_IF

			IF COM.bMoveBusy THEN
				COM.inUSe 	:= TRUE;
			ELSE
				COM.inUSe 	:= FALSE;
			END_IF
			
			IF COM.bMoveDone THEN
				COM.bEnable := FALSE;
				COM.bCouple := FALSE;
				COM.inUSe 	:= FALSE;
				COM.bMoveX 	:= FALSE;
				COM.bMoveY 	:= FALSE;
				COM.bMoveZ 	:= FALSE;
				index 	:= 0;
			END_IF
		ELSE
			index 	:= 995;
		END_IF
		
	205: //Go to xy Pos
    	COM.absX := (COM.goX);
		COM.absY := (COM.goY);
		
		IF gvl.configHoming THEN
			COM.bEnable := TRUE;
			COM.bCouple := TRUE;
			
			IF wait100ms.Q THEN 
				COM.bMoveX 	:= TRUE;
				COM.bMoveY 	:= TRUE;
			END_IF
			
			IF COM.bMoveBusy THEN
				COM.inUSe 	:= TRUE;
			ELSE
				COM.inUSe 	:= FALSE;
			END_IF
			
			IF COM.bMoveXDone AND COM.bMoveYDone THEN
				COM.bEnable := FALSE;
				COM.bCouple := FALSE;
				COM.inUSe 	:= FALSE;
				COM.bMoveX 	:= FALSE;
				COM.bMoveY 	:= FALSE;
				COM.bMoveZ 	:= FALSE;
				index 	:= 0;
			END_IF
		ELSE
			index 	:= 995;
		END_IF
		
	210: //Go X Pos
	    COM.absX := (com.goX);
		
		IF gvl.configHoming THEN
			COM.bEnable := TRUE;
			COM.bCouple := TRUE;
		
			IF wait100ms.Q THEN 
				COM.bMoveX 	:= TRUE;
			END_IF
			
			IF COM.bMoveBusy THEN
				COM.inUSe 	:= TRUE;
			ELSE
				COM.inUSe 	:= FALSE;
			END_IF
			
			IF COM.bMoveXDone THEN
				COM.bEnable := FALSE;
				COM.bCouple := FALSE;
				COM.inUSe 	:= FALSE;
				COM.bMoveX 	:= FALSE;
				index 	:= 0;
			END_IF
		ELSE
			index 	:= 995;
		END_IF
		
	220: //Go Y Pos
		COM.absY := (com.goY);
		
		IF gvl.configHoming THEN
			COM.bEnable := TRUE;
			
			IF wait100ms.Q THEN 
				COM.bMoveY 	:= TRUE;
			END_IF
					
			IF COM.bMoveBusy THEN
				COM.inUSe 	:= TRUE;
			ELSE
				COM.inUSe 	:= FALSE;
			END_IF
			
			IF COM.bMoveYDone THEN
				COM.bEnable := FALSE;
				COM.bCouple := FALSE;
				COM.inUSe 	:= FALSE;
				COM.bMoveY 	:= FALSE;
				index 	:= 0;
			END_IF
		ELSE
			index 	:= 995;
		END_IF
			
	230: //Go Z Pos
		COM.absZ := (com.goZ);
		
		IF gvl.configZaxis THEN
			COM.bEnable := TRUE;
			
			IF wait100ms.Q THEN 
				COM.bMoveZ 	:= TRUE;
			END_IF
			
			IF COM.bMoveBusy THEN
				COM.inUSe 	:= TRUE;
			ELSE
				COM.inUSe 	:= FALSE;
			END_IF
			
			IF COM.bMoveZDone THEN
				COM.bEnable := FALSE;
				COM.bCouple := FALSE;
				COM.inUSe 	:= FALSE;
				COM.bMoveZ 	:= FALSE;
				index 	:= 0;
			END_IF
		ELSE
			index := 996;
		END_IF
		
	250: //Execute Gcode
		GVL.message_pub  := '{"text": "Executing code say reset after the program"}';
		GVL.bSendMessage := TRUE;
		
		IF gvl.configHoming AND FALSE THEN
			COM.bEnable := TRUE;
			gcode.bBuildGroup := TRUE;
			gcode.bLoad := TRUE;
						
			IF wait100ms.Q THEN 
				gcode.bStart 	:= TRUE;
				gcode.bLoad := FALSE;
			ELSE 
				gcode.bStart 	:= FALSE;
			END_IF
			
			IF 	(command = 'reset' OR command = 'stop') THEN
				gcode.bStop	:= TRUE;
				gcode.bReset := TRUE;
				gcode.bBuildGroup := FALSE;
				COM.bEnable := FALSE;
				
			ELSIF(gcode.bStop)THEN
					gcode.bStop	:= FALSE;
					gcode.bReset := FALSE;
					COM.bEnable := FALSE;
					
					index 		:= 0;
			END_IF
			
		ELSE
			index := 995;
		END_IF
			
	260: //execute trace
		GVL.message_pub  := '{"text": "Tracing will be executed"}';
		GVL.bSendMessage := TRUE;
		index 		:= 0;
		
	270: //execute sort
		GVL.message_pub  := '{"text": "executing sort"}';
		GVL.bSendMessage := TRUE;
		index 		:= 0;
		
	280: //execute drill
		GVL.message_pub  := '{"text": "execute drill"}';
		GVL.bSendMessage := TRUE;
		index 		:= 0;
		
	300: //Read XYZ
		actualX 	:= COM.PosX;
		actualY 	:= COM.Posy;
		actualZ 	:= COM.PosZ;
		IF COM.bValid THEN
			index 	:= 0;
		END_IF
	
	450: //Up
		COM.relZ := (-com.goZ);
		COM.bEnable := TRUE;
		
		IF wait100ms.Q THEN 
			COM.bRelZ 	:= TRUE;
		END_IF
		
		IF COM.bMoveBusy THEN
			COM.inUSe 	:= TRUE;
		ELSE
			COM.inUSe 	:= FALSE;
		END_IF
		
		IF COM.bMoveZRelDone THEN
			COM.bEnable := FALSE;
			COM.bCouple := FALSE;
			COM.inUSe 	:= FALSE;
			COM.brelZ 	:= FALSE;
			index 	:= 0;
		END_IF	
	
	460: //Down
		COM.relZ := (com.goZ);
		COM.bEnable := TRUE;
		
		IF wait100ms.Q THEN 
			COM.bRelZ 	:= TRUE;
		END_IF
		
		IF COM.bMoveBusy THEN
			COM.inUSe 	:= TRUE;
		ELSE
			COM.inUSe 	:= FALSE;
		END_IF
		
		IF COM.bMoveZRelDone THEN
			COM.bEnable := FALSE;
			COM.bCouple := FALSE;
			COM.inUSe 	:= FALSE;
			COM.brelZ 	:= FALSE;
			index 	:= 0;
		END_IF
			
	600: //Show object
		com.objectNum := com.object1;
		com.readfile  := TRUE;

		
		IF gvl.configHoming THEN
			COM.bEnable := TRUE;
			COM.bCouple := TRUE;
			
			IF wait100ms.Q THEN 
				COM.absX := LREAL_TO_INT(COM.objectx);
				COM.absY := LREAL_TO_INT(COM.objecty);
				com.objectread := TRUE;
			END_IF
			
			IF wait200ms.Q THEN 
				COM.bMoveX 	:= TRUE;
				COM.bMoveY 	:= TRUE;
				com.objectread := FALSE;
			END_IF
			
			IF COM.bMoveBusy THEN
				COM.inUSe 	:= TRUE;
			ELSE
				COM.inUSe 	:= FALSE;
			END_IF
			
			IF COM.bMoveXDone AND COM.bMoveYDone THEN
				COM.bEnable := FALSE;
				COM.bCouple := FALSE;
				COM.inUSe 	:= FALSE;
				COM.bMoveX 	:= FALSE;
				COM.bMoveY 	:= FALSE;
				COM.bMoveZ 	:= FALSE;
				index 	:= 0;
			END_IF
		ELSE
			index 	:= 995;
		END_IF
	

	996: //set z to zero before performing an action on the z axis
		GVL.message_pub  := '{"text": "You have to do Z to zero first"}';
		GVL.bSendMessage := TRUE;
		index := 0;
	999: //Error
			COM.bEnable := FALSE;
			gvl.StopALL := TRUE;
			GVL.message_pub  := '{"text": "There has been an error use reset command"}';
			GVL.bSendMessage := TRUE;
			IF(command = 'reset')THEN
				gvl.StopALL := FALSE;
				index := 0;
			END_IF

	ELSE 
		index := 0;
END_CASE;

END_PROGRAM

// ---- POUs/COMMANDS/commandExecute.TcPOU
PROGRAM commandExecute
VAR
	MCPower_Xa, MCPower_Xb, MCPower_Y, 	MCPower_Z 	: MC_Power;
	MCResetXa, MCResetXb, MCResetY, MCResetZ		: MC_Reset;

	fb_MCGearIn										: MC_GearIn;
	fb_MCGearOut									: MC_GearOut;

	fb_MCHOME_X, fb_MCHOME_Y						: MC_Home;
	fb_MoveAbs_X, fb_MoveAbs_Y, fb_MoveAbs_Z 		: MC_MoveAbsolute;
	fb_MoveRel_Z 									: MC_MoveRelative;
	fb_ReadX, fb_ReadY, fb_readZ 					: MC_ReadActualPosition;

	fb_SetZToZero 									: MC_SetPosition;
END_VAR

//Enable Axis
	MCPower_Xa(
		Axis	:= GVL.As_Xa, 
		Enable	:= COM.bEnable, 
		Enable_Positive:= COM.bEnable, 
		Enable_Negative:= COM.bEnable, 
		Override:= 100 );
		
	MCPower_Xb(
		Axis	:= GVL.As_Xb, 
		Enable	:= COM.bEnable, 
		Enable_Positive:= COM.bEnable, 
		Enable_Negative:= COM.bEnable, 
		Override:= 100 );
		
	MCPower_Y(
		Axis	:= GVL.As_Y, 
		Enable	:= COM.bEnable, 
		Enable_Positive:= COM.bEnable, 
		Enable_Negative:= COM.bEnable, 
		Override:= 100 );
		
	MCPower_Z(
		Axis	:= GVL.As_Z, 
		Enable	:= COM.bEnable, 
		Enable_Positive:= COM.bEnable, 
		Enable_Negative:= COM.bEnable, 
		Override:= 100 );

//Reset Axis
	MCResetXa(
		Axis	:= GVL.As_Xa, 
		Execute	:= COM.bReset );
	
	MCResetXb(
		Axis	:= GVL.As_Xb, 
		Execute	:= COM.bReset );

	MCResetY(
		Axis	:= GVL.As_Y, 
		Execute	:= COM.bReset );

	MCResetZ(
		Axis	:= GVL.As_Z, 
		Execute	:= COM.bReset );
	
//Couple Axis
	fb_MCGearIn(
		Master	:= GVL.As_Xa, 
		Slave	:= GVL.As_Xb, 
		Execute := COM.bCouple, 
		RatioNumerator:= 1, 
		RatioDenominator:= 1 );
		
	fb_MCGearOut(
		Slave	:= GVL.As_Xb,
		Execute := NOT(COM.bCouple) );
		
//Homing
	fb_MCHOME_X(
		Axis     := GVL.As_Xa, 
		Execute  := COM.bHome AND COM.bCouple, 
		Position := 0, 
		bCalibrationCam:= GVL.bX1 );
	
	fb_MCHOME_Y(
		Axis	 := GVL.As_Y, 
		Execute  := COM.bHome AND COM.bCouple, 
		Position := 0, 
		bCalibrationCam:= GVL.bY1 );
		
//Absolute movement
	fb_MoveAbs_X(
		Axis 	 := GVL.As_Xa,
		Execute  := COM.bMoveX AND COM.bCouple,
		Position := COM.absX,
		Velocity := COM.velX);
		
	fb_MoveAbs_Y(
		Axis 	 := GVL.As_Y,
		Execute  := COM.bMoveY,
		Position := COM.absY,
		Velocity := COM.velY);		
		
	fb_MoveAbs_Z(
		Axis 	 := GVL.As_Z,
		Execute  := COM.bMoveZ,
		Position := COM.absZ,
		Velocity := COM.velZ);
//Rel movement
	fb_MoveRel_Z(
		Axis 	 := GVL.As_Z,
		Execute  := COM.bRelZ,
		distance := COM.relZ,
		Velocity := COM.velZ);			
		
//set Z postition to zero
	fb_SetZToZero(
		Axis := GVL.As_Z, 
		Execute := COM.bSetZ,
		Position := 0, 
		Mode := FALSE);

//read actual position
	fb_ReadX(Enable := TRUE, Axis := GVL.As_Xa, Position => COM.PosX);
	fb_ReadY(Enable := TRUE, Axis := GVL.As_Y, Position => COM.PosY);
	fb_ReadZ(Enable := TRUE, Axis := GVL.As_Z, Position => COM.PosZ);
	COM.bValid := fb_ReadX.Valid AND fb_ReadY.Valid AND fb_ReadZ.Valid;
	
//done = busy
	COM.bHomeBusy	:= fb_MCHOME_X.Busy OR fb_MCHOME_Y.Busy;
	COM.bMoveBusy	:= fb_MoveAbs_X.Busy OR fb_MoveAbs_Y.Busy OR fb_MoveAbs_Z.Busy;		
	
	COM.bHomeDone	:= fb_MCHOME_X.Done AND fb_MCHOME_Y.Done;
	COM.bMoveDone	:= fb_MoveAbs_X.Done AND fb_MoveAbs_Y.Done AND fb_MoveAbs_Z.Done;
	
	COM.bMoveXDone	:= fb_MoveAbs_X.Done;
	COM.bMoveYDone	:= fb_MoveAbs_Y.Done;
	COM.bMoveZDone	:= fb_MoveAbs_Z.Done;
	COM.bMoveZRelDone	:= fb_MoveRel_Z.Done;

END_PROGRAM

// ---- POUs/MQTT/MAIN_MQTT.TcPOU
PROGRAM MAIN_MQTT
VAR
	
	arr : ARRAY [1..10] OF STRING(2047);
	
	(* JSON *)
	fbJson 			: FB_JsonDomParser;
	jsonDoc 		: SJsonValue;
	jsonProp		: SJsonValue;
	jsonValue		: SJsonValue;
	bHasMember		: BOOL;
	stReceivedData	: STRING(255);
	stReceivedData_arr : ARRAY [1..10] OF STRING(255);
	
	(* Test *)
	test			: STRING(255);
	test_recv		: STRING(255);
	
	teller: INT := 0;
END_VAR

IF NOT (GVL.flag_pub) THEN
	PrgMqttCom();
	SubMqttCom();
END_IF

//Pub to text_to_speech--------------------------------------------------------------------
IF GVL.flag_pub AND GVL.bSendMessage THEN
	//GVL.message_pub := '{"text": "This is a test"}';
	PrgMqttCom();
	GVL.message_pub := '';
	GVL.bSendMessage := FALSE;
END_IF

SubMqttCom();

END_PROGRAM

// ---- POUs/MQTT/PrgMqttCom.TcPOU
PROGRAM PrgMqttCom
VAR
	fbMqttClient : FB_IotMqttClient;
	bSetParameter : BOOL := TRUE;
	bConnect : BOOL := TRUE;
	
	(* published message *)
	sTopicPub : STRING(255) := 'Test/Text_To_Speech';
	sPayloadPub : STRING(255);
	
	hrErrorOccurred : HRESULT; // contains the latest occurred error
END_VAR

IF bSetParameter THEN
	bSetParameter := FALSE;
	fbMqttClient.sHostName:= '192.168.1.205';
	fbMqttClient.nHostPort:= 1883;
	fbMqttClient.sTopicPrefix:= ''; 
END_IF

sPayloadPub := GVL.message_pub;

IF NOT(GVL.flag_pub) THEN
	fbMqttClient.Execute(bConnect);
	IF fbMqttClient.bError THEN
		hrErrorOccurred := fbMqttClient.hrErrorCode;
	END_IF
	IF fbMqttClient.bConnected THEN
		GVL.flag_pub := TRUE;
	END_IF
END_IF

IF GVL.flag_pub THEN
		fbMqttClient.Publish(	sTopic:= sTopicPub, 
								pPayload:= ADR(sPayloadPub), nPayloadSize:= LEN2(ADR(sPayloadPub)), 
								eQoS:= TcIotMqttQos.AtMostOnceDelivery, bRetain:= FALSE, bQueue:= FALSE );
		IF fbMqttClient.bError THEN
			hrErrorOccurred := fbMqttClient.hrErrorCode;
		END_IF
END_IF

END_PROGRAM

// ---- POUs/MQTT/SubMqttCom.TcPOU
PROGRAM SubMqttCom
VAR
	fbMqttClient : FB_IotMqttClient;
	bSetParameter : BOOL := TRUE;
	bConnect : BOOL := TRUE;
	
	(* received message *)
	bSubscribed : BOOL;
	sTopicSub : STRING(255) := 'hermes/intent/GeneraalAlfa:PLC';//GeneraalAlfa:machineState
	{attribute 'TcEncoding':='UTF-8'}
	sTopicRcv : STRING(255);
	{attribute 'TcEncoding':='UTF-8'}
	sPayloadRcv : STRING(2047);
	sPayloadRcv_extra : STRING(2047);
	fbMessageQueue : FB_IotMqttMessageQueue;
	fbMessage : FB_IotMqttMessage;
	
	hrErrorOccurred : HRESULT; // contains the latest occurred error
END_VAR

IF bSetParameter THEN
	bSetParameter := FALSE;
	fbMqttClient.sHostName:= '192.168.1.205';
	fbMqttClient.nHostPort:= 1883;
	fbMqttClient.sTopicPrefix:= ''; 
	fbMqttClient.ipMessageQueue := fbMessageQueue;
END_IF

fbMqttClient.Execute(bConnect);
IF fbMqttClient.bError THEN
	hrErrorOccurred := fbMqttClient.hrErrorCode;
END_IF

IF fbMessageQueue.nQueuedMessages > 0 THEN
	IF fbMessageQueue.Dequeue(fbMessage:=fbMessage) THEN
		fbMessage.GetTopic(pTopic:=ADR(sTopicRcv), nTopicSize:=SIZEOF(sTopicRcv) );
		fbMessage.GetPayload(pPayload:=ADR(sPayloadRcv), nPayloadSize:=SIZEOF(sPayloadRcv), bSetNullTermination:=FALSE);
	END_IF
END_IF

IF fbMqttClient.bConnected THEN
	IF NOT bSubscribed THEN
		bSubscribed := fbMqttClient.Subscribe(sTopic:=sTopicSub, eQoS:=TcIotMqttQos.AtMostOnceDelivery);
		IF fbMqttClient.bError THEN
			hrErrorOccurred := fbMqttClient.hrErrorCode;
		END_IF
	END_IF
END_IF

IF NOT( sPayloadRcv = '')THEN
	sPayloadRcv_extra := sPayloadRcv;
	GVL.message_sub := sPayloadRcv;
	sPayloadRcv :='';
END_IF

END_PROGRAM

// ---- POUs/COMMANDS/POU_NCI.TcPOU
PROGRAM POU_NCI
VAR
	fb_BuildGroup: CfgBuild3DGroup;
	fb_ReconfigGroup: CfgReconfigGroup;
	fb_LoadProg: ItpLoadProgEx;
	fb_StartStop: ItpStartStopEx;
	fb_Reset: ItpResetEx2;
	
END_VAR

fb_BuildGroup(
	bExecute:= gcode.bBuildGroup, 
	nGroupId:= GVL.ChannelInput.GrpId, 
	nXAxisId:= GVL.As_Xa.NcToPlc.AxisId, 
	nYAxisId:= GVL.As_Y.NcToPlc.AxisId, 
	nZAxisId:= GVL.As_Z.NcToPlc.AxisId, 
	tTimeOut:= T#1S );
	
fb_ReconfigGroup(
	bExecute:= NOT(gcode.bBuildGroup), 
	nGroupId:= GVL.ChannelInput.GrpId, 
	tTimeOut:= T#1S );
	
ItpSetOverridePercent(fOverridePercent:= 100, sPlcToNci:= GVL.ChannelOutput);

fb_LoadProg(
	sNciToPlc:= GVL.ChannelInput, 
	bExecute:= gcode.bLoad, 
	sPrg:= '\HARD DISK\TWINCAT\Mc\Nci\Gcode_test1.nc', 
	nLength:= LEN('\HARD DISK\TWINCAT\Mc\Nci\Gcode_test1.nc'), 
	tTimeOut:= T#1S );
	
fb_StartStop(
	bStart:= gcode.bStart, 
	bStop:= gcode.bStop OR gvl.StopALL, 
	tTimeOut:= T#1S, 
	sNciToPlc:= GVL.ChannelInput );
	
fb_Reset(
	bExecute:= gcode.bReset, 
	tTimeOut:= T#1S, 
	sNciToPlc:= GVL.ChannelInput );

END_PROGRAM

// ---- POUs/JSON/decCOM_PLC.TcPOU
PROGRAM decCOM_PLC
VAR
	 recString 			: STRING(2047);
	 RisingEdge         : R_TRIG;
	 bExecute			: BOOL;
	 bReset				: BOOL;

	fbJson 				: FB_JsonDomParser;
                    	
	jsonDoc 			: SJsonValue;
	jsonDoc2 			: SJsonValue;
	                	
	jsonProp			: SJsonValue;
	jsonProp2			: SJsonValue;           	

	jsontempval			: SJsonValue;
	
	getInput			: STRING(2047);
	getRawValue 		: STRING;
	getValueStr 		: STRING;
	getValue1			: STRING(2047);
	
	jsonGetulint		: ULINT;
	jsongettype			: Tc3_JsonXml.EJsonType;
	jsongetArraySize	: UDINT;
	jsongetArray		: ARRAY[0..1000] OF SJsonValue;
	jsongetArrayulint	: ULINT;
	jsongetArrayudint	: UDINT;
	
	JSONTEMP			: STRING(2047);
	
	JSONVal1 			: STRING;
	JSONVal2 			: STRING;
	JSONVal3 			: STRING;
	JSONVal4 			: STRING;
	JSONVal5 			: STRING;
	JSONVal6 			: STRING;
	
	cnt : UDINT;	
	temp : string;
END_VAR

RisingEdge(CLK:=bReset);
IF RisingEdge.Q THEN
	JSONVal1	:= '';
	JSONVal2	:= '';
	JSONVal3	:= '';
    JSONVal4	:= '';
    JSONVal5	:= '';
    JSONVal6	:= '';
	bReset 		:= FALSE;
END_IF

IF NOT(GVL.message_sub = '') THEN
	recString := GVL.message_sub;
	jsonDoc := fbJson.ParseDocument(recString);
	
	jsonProp := fbJson.FindMember(jsonDoc, 'slots');
	cnt := 0;
	
	IF (jsonProp <> 0) THEN
		jsongettype			:= fbJson.GetType(jsonProp);
		jsongetArraySize	:= fbJson.GetArraySize(jsonProp);
		FOR cnt := 0 TO jsongetArraySize-1 BY 1 DO
			jsongetArrayudint		:= fbJson.GetArrayValueByIdx(jsonProp, cnt);
			JSONTEMP				:= fbJson.GetJson( jsongetArrayudint );
				jsonDoc2 			:= fbJson.ParseDocument(JSONTEMP);
				jsonProp2 			:= fbJson.FindMember(jsonDoc2, 'value');
					jsonProp2 		:= fbJson.FindMember(jsonProp2, 'value');
						CASE cnt OF
							0:	JSONVal1	:= fbJson.GetString(jsonProp2);
							1:	JSONVal2	:= fbJson.GetString(jsonProp2);
							2:	JSONVal3	:= fbJson.GetString(jsonProp2);
							3:	JSONVal4	:= fbJson.GetString(jsonProp2);
							4:	JSONVal5	:= fbJson.GetString(jsonProp2);
							5:	JSONVal6	:= fbJson.GetString(jsonProp2);
						END_CASE
		END_FOR
		
		CASE cnt OF
			1:
				IF 		(JSONVal1 = 'Do homing') 						THEN							com.sendCommand := 'do homing';				
				ELSIF 	(JSONVal1 = 'Execute trace') 					THEN							com.sendCommand := 'execute trace';			
				ELSIF 	(JSONVal1 = 'Execute sort') 					THEN							com.sendCommand := 'execute sort';
				ELSIF 	(JSONVal1 = 'Execute Drill') 					THEN							com.sendCommand := 'execute drill';
				ELSIF 	(JSONVal1 = 'Stop') 							THEN							com.sendCommand := 'stop';	
				ELSIF 	(JSONVal1 = 'z to zero') 						THEN							com.sendCommand := 'z to zero';
				ELSIF 	(JSONVal1 = 'read position') 					THEN							com.sendCommand := 'read position';	
				ELSIF 	(JSONVal1 = 'read error') 						THEN							com.sendCommand := 'read error';	
				ELSIF 	(JSONVal1 = 'read files') 						THEN							com.sendCommand := 'read files';	
				ELSIF 	(JSONVal1 = 'execute Gcode')					THEN							com.sendCommand := 'execute gcode';	
				ELSIF 	(JSONVal1 = 'reset') 							THEN							com.sendCommand := 'reset';	
				END_IF
			2:
				IF 		(JSONVal1 = 'show difference') 					THEN							com.sendCommand := 'show difference';
																										com.object1		:= STRING_TO_INT(JSONVal2);	
				ELSIF 	(JSONVal1 = 'show object') 						THEN							com.sendCommand := 'show object';
																										com.object1		:= STRING_TO_INT(JSONVal2);	
				ELSIF 	(JSONVal1 = 'delete difference') 				THEN							com.sendCommand := 'delete difference';
																										com.object1		:= STRING_TO_INT(JSONVal2);	
				ELSIF 	(JSONVal1 = 'turn difference') 					THEN							com.sendCommand := 'turn difference';
																										com.object1		:= STRING_TO_INT(JSONVal2);
				ELSIF 	(JSONVal1 = 'turn object') 						THEN							com.sendCommand := 'turn object';
																										com.object1		:= STRING_TO_INT(JSONVal2);
				ELSIF 	(JSONVal1 = 'X-axis') 							THEN							com.sendCommand := 'x-axis';
																										com.goX		:= STRING_TO_INT(JSONVal2);
				ELSIF 	(JSONVal1 = 'Y-axis') 							THEN							com.sendCommand := 'y-axis';
																										com.goY		:= STRING_TO_INT(JSONVal2);
				ELSIF 	(JSONVal1 = 'Z-axis') 							THEN							com.sendCommand := 'z-axis';
																										com.goZ		:= STRING_TO_INT(JSONVal2);
				ELSIF 	(JSONVal1 = 'Up') 								THEN							com.sendCommand := 'Up';
																										com.goZ		:= STRING_TO_INT(JSONVal2);
				ELSIF 	(JSONVal1 = 'Down') 							THEN							com.sendCommand := 'Down';
																										com.goZ		:= STRING_TO_INT(JSONVal2);					
				END_IF
			4:
				IF 		(JSONVal1 = 'X-axis' AND JSONVal3 = 'Y-axis')	THEN 							com.sendCommand := 'go xy';
																										com.goX			:= STRING_TO_INT(JSONVal2);	
																										com.goY			:= STRING_TO_INT(JSONVal4);		
				ELSIF 	(JSONVal1 = 'combine difference') 				THEN							com.sendCommand := 'combine difference';
																										com.object1		:= STRING_TO_INT(JSONVal2);	
																										com.object2		:= STRING_TO_INT(JSONVal4);
				ELSIF 	(JSONVal1 = 'combine object') 					THEN							com.sendCommand := 'combine object';
																										com.object1		:= STRING_TO_INT(JSONVal2);	
																										com.object2		:= STRING_TO_INT(JSONVal4);
				END_IF													
			6:
				IF 		(JSONVal1 = 'X-axis' AND JSONVal3 = 'Y-axis' AND JSONVal5 = 'Z-axis') THEN		com.sendCommand := 'go xyz';
																										com.goX			:= STRING_TO_INT(JSONVal2);	
																										com.goY			:= STRING_TO_INT(JSONVal4);
																										com.goZ			:= STRING_TO_INT(JSONVal6);
				END_IF
		END_CASE
	END_IF
	GVL.message_sub := '';
	temp := recString;
	recString := '';
END_IF

END_PROGRAM

// ---- POUs/knoppen.TcPOU
PROGRAM knoppen
VAR
	bmagneet	    AT %Q* : BOOL;
	bpomp1			AT %Q* : BOOL;
	bpomp2			AT %Q* : BOOL;
END_VAR

END_PROGRAM

// ---- GlobalTextList.TcGTLO
TEXTLIST GlobalTextList
  943 = 'Absolute'
  163 = 'Couple'
  730 = 'Group'
  610 = 'Home'
  23 = 'Load'
  962 = 'magneet'
  172 = 'move abs X'
  424 = 'Move abs X'
  68 = 'move abs Y'
  700 = 'Move abs Y'
  459 = 'move ABS z'
  52 = 'move abs z'
  760 = 'move abs Z'
  258 = 'Move abs Z'
  193 = 'move rel X'
  135 = 'Move rel X'
  829 = 'move rel Y'
  787 = 'Move rel Y'
  698 = 'move rel z'
  917 = 'move rel Z'
  750 = 'Move rel z'
  793 = 'Niet gebruiken'
  57 = 'pomp1'
  216 = 'pomp2'
  769 = 'Reconfig'
  653 = 'Relative'
  187 = 'Reset'
  285 = 'set z on pos 0'
  244 = 'Set Z pos to 0'
  127 = 'Start'
  887 = 'Stop'
  966 = 'STOP'
END_TEXTLIST

// ---- VISUs/Basic.TcVIS
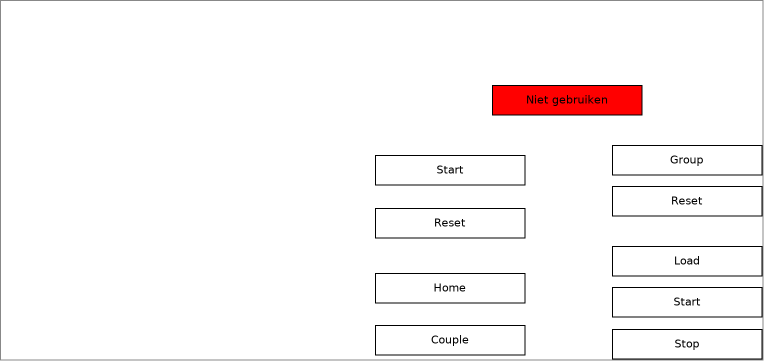
VISUALIZATION Basic  // 764x361
    Rectangle (375,325 150x30), "Couple", colour toggle: INIT.bGearIn
        toggle INIT.bGearIn
    Rectangle (375,273 150x30), "Home"
        tap INIT.bHome
    Rectangle (375,155 150x30), "Start", colour toggle: INIT.bEN
        toggle INIT.bEN
    Rectangle (375,208 150x30), "Reset", colour toggle: INIT.bReset
        tap INIT.bReset
    Rectangle (612,145 150x30), "Group", colour toggle: POU_NCI.bBuildGroup
        toggle POU_NCI.bBuildGroup
    Rectangle (612,186 150x30), "Reset"
        tap POU_NCI.bReset
    Rectangle (612,287 150x30), "Start"
        tap POU_NCI.bStart
    Rectangle (612,329 150x30), "Stop"
        tap POU_NCI.bStop
    Rectangle (612,246 150x30), "Load"
        tap POU_NCI.bLoad
    Rectangle (492,85 150x30), "Niet gebruiken"
END_VISUALIZATION

// ---- VISUs/bStopAll.TcVIS
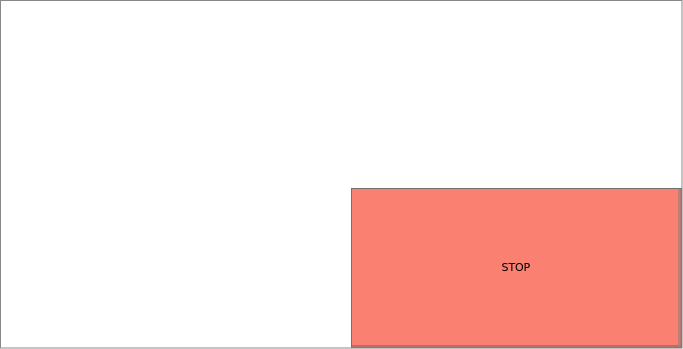
VISUALIZATION bStopAll  // 683x349
    Button (351,188 330x159), "STOP", colour toggle: GVL.StopALL
        toggle GVL.StopALL
END_VISUALIZATION

// ---- VISUs/vKnoppen.TcVIS
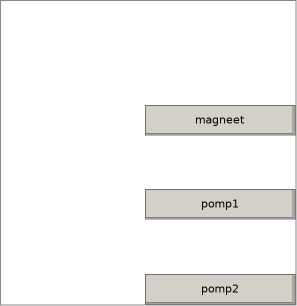
VISUALIZATION vKnoppen  // 297x306
    Button (145,105 150x30), "magneet", colour toggle: knoppen.bmagneet
        toggle knoppen.bmagneet
    Button (145,189 150x30), "pomp1", colour toggle: knoppen.bpomp1
        toggle knoppen.bpomp1
    Button (145,274 150x30), "pomp2", colour toggle: knoppen.bpomp2
        toggle knoppen.bpomp2
END_VISUALIZATION
